// TIA Portal V17 export
// export: Created 2022-07-20T07:02:38.7958792Z, ExportSetting WithDefaults, DisplayName Totally Integrated Automation Portal, DisplayVersion V17, DisplayName TIA Portal Openness, DisplayVersion V17, DisplayName TIA Portal Version Control Interface, DisplayVersion V17, DisplayName SINAMICS Startdrive Advanced, DisplayVersion V17, DisplayName SINAMICS Startdrive G130, G150, S120, S150, SINAMICS MV, S210, DisplayVersion V17, DisplayName SINAMICS Startdrive G110M, G120, G120C, G120D, G120P, G115D, DisplayVersion V17, DisplayName STEP 7 Professional, DisplayVersion V17, DisplayName STEP 7 Safety, DisplayVersion V17, DisplayName WinCC Advanced, DisplayVersion V17
VAR_GLOBAL   // PLC tag table "IFM_BeaconTower_CommunicationTable"
   BeaconTower1_IFM_OutWord_0 AT %QW506 : Word;
   BeaconTower1_IFM_OutWord_2 AT %QW508 : Word;
   BeaconTower1_IFM_OutWord_4 AT %QW510 : Word;
   BeaconTower1_IFM_OutWord_6 AT %QW512 : Word;
END_VAR
